(* CoDeSys 2.3.9.52 project: UseOfFunctionBlock_Template.pro *)
(* Libraries: STANDARD.LIB*16.8.17 14:08:57 *)

(* POU MAIN, ST *)
PROGRAM MAIN
VAR
	fbInst_1	: FB_Example;	(* 1st instance *)
	fbInst_2	: FB_Example;	(* 2nd instance *)
	bCalling	: BOOL :=TRUE;	(*Calling instance vs. assigining values*)
	btnIn		: BOOL;			(*InputButton*)
END_VAR
(*Calling instance nbr 1*)
fbInst_1(
	bReset:= ,
	bIn:= ,
	bOut=> ,
	iC_trig=> ,
	iC_run=> );

(*Using instance nbr 2*)
IF bCalling THEN
	(*Calling instance nbr 2. Use btnIn to control the bIn of instance*)
	;
ELSE
	(*Assigning instance nbr 2 values. Use btnIn to control the bIn of instance*)
	;
END_IF;
END_PROGRAM

(* POU FB_Example, ST *)
FUNCTION_BLOCK FB_Example
VAR_INPUT
	bReset	: BOOL;	(*Reset signal*)
	bIn		: BOOL;	(*Input trigger from user*)
END_VAR
VAR_OUTPUT
	bOut	: BOOL;	(*Output state*)
	iC_trig	: UINT;	(*Counter for triggered signals*)
	iC_run	: UINT;	(*Running counter*)
END_VAR
VAR
	rTrig_In	: R_TRIG;	(*Rising trigger for input*)
END_VAR
(*Reset handler: Reset counters and outputs, if reset is requested*)


(*Rising edge is provided?*)
rTrig_In(CLK:= , Q=> );

(*Increase trigger counter once per pressing IN -button*)

(*Increase running counter. Once per PLC cycle*)

(*Set output according user input*)
END_FUNCTION_BLOCK

(* Visualisation VC_FB_Example
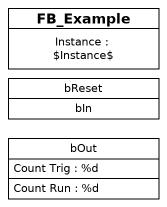
rectangle at (0,150)-(151,171): text "Count Trig : %d"; shows $FB$.iC_trig
rectangle at (0,0)-(151,21): text "FB_Example"
rectangle at (0,20)-(151,61): text "Instance : / $Instance$"
rounded rectangle at (0,70)-(151,91): text "bReset"; alarm colour if $FB$.bReset; taps $FB$.bReset
rounded rectangle at (0,90)-(151,111): text "bIn"; alarm colour if $FB$.bIn; taps $FB$.bIn
rectangle at (0,130)-(151,151): text "bOut"; alarm colour if $FB$.bOut
rectangle at (0,170)-(151,191): text "Count Run : %d"; shows $FB$.iC_run
*)

(* Visualisation VC_MAIN_Panel
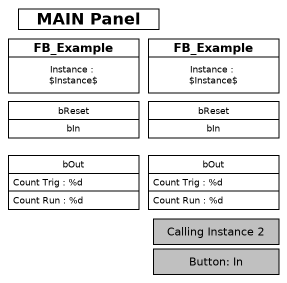
rectangle at (10,0)-(151,21): text "MAIN Panel"
embedded screen at (0,30)-(131,201): VC_FB_Example
embedded screen at (140,30)-(271,201): VC_FB_Example
rounded rectangle at (145,210)-(271,236): text "Calling Instance 2"; alarm colour if MAIN.bCalling; toggles MAIN.bCalling
rounded rectangle at (145,240)-(271,266): text "Button: In"; alarm colour if MAIN.btnIn; taps MAIN.btnIn
*)
